(* CoDeSys 2.3.9.41 project: lek_obyav.pro *)
(* Libraries: Standard.lib 4.10.05 11:14:46, IecSfc.lib 13.4.06 15:51:28, SYSLIBCALLBACK.LIB 26.9.08 16:43:52 *)

(* POU PLC_PRG, ST *)
PROGRAM PLC_PRG
VAR

	tim1 : TIME ;
	Temp_vozduha : INT := -10; (*Температура воздуха*)
	Nasos1 , Vent , Klapan : BOOL ;

END_VAR
VAR RETAIN

	Mess1 : STRING := 'Пожар';

END_VAR
;
END_PROGRAM
